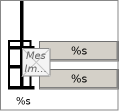
VISUALIZATION VISU_VERIN_VH  // 119x111
VAR_IN_OUT
	m_Input_VERIN: BLOCK_ACTUATOR;
	m_Input_MAINT: BOOL;
END_VAR
    Rectangle (8,40 23x49)
    Group (9,1 23x46), invisible if: NOT m_Input_VERIN.STATE_On
        Rectangle (0,45 25x3)
        Rectangle (11,0 3x47)
    Group (9,20 23x46), invisible if: (m_Input_VERIN.STATE_ON OR m_Input_VERIN.STATE_OFF) <> 0
        Rectangle (0,45 25x3)
        Rectangle (11,0 3x47)
    Group (9,41 23x46), invisible if: NOT m_Input_VERIN.STATE_OFF
        Rectangle (0,45 25x3)
        Rectangle (11,0 3x47)
    Rectangle (1,91 45x20), "%s", text variable: m_Input_VERIN.MNEMO
    Button (39,41 80x20), "%s", invisible if: NOT m_Input_VERIN.AUTOR_On_IHM OR NOT m_Input_MAINT, input disabled if: NOT m_Input_VERIN.AUTOR_On_IHM OR NOT m_Input_MAINT, text list: 'TextList_Orders', text index: 3
        tap m_Input_VERIN.M_On
    Button (39,69 80x20), "%s", invisible if: NOT m_Input_VERIN.AUTOR_Off_IHM OR NOT m_Input_MAINT, input disabled if: NOT m_Input_VERIN.AUTOR_Off_IHM OR NOT m_Input_MAINT, text list: 'TextList_Orders', text index: 2
        tap m_Input_VERIN.M_Off
    Image (22,48 28x28), invisible if: NOT m_Input_VERIN.STATE_NOK, image: MesImages.warning
END_VISUALIZATION

(* stored: Version 1.1.0.1, ProductVersion 3.1.4024.10
   Visu VISU_VERIN_VH: Id {78a7b077-e4fd-4eea-bd3e-d15e1f195c2a} *)
